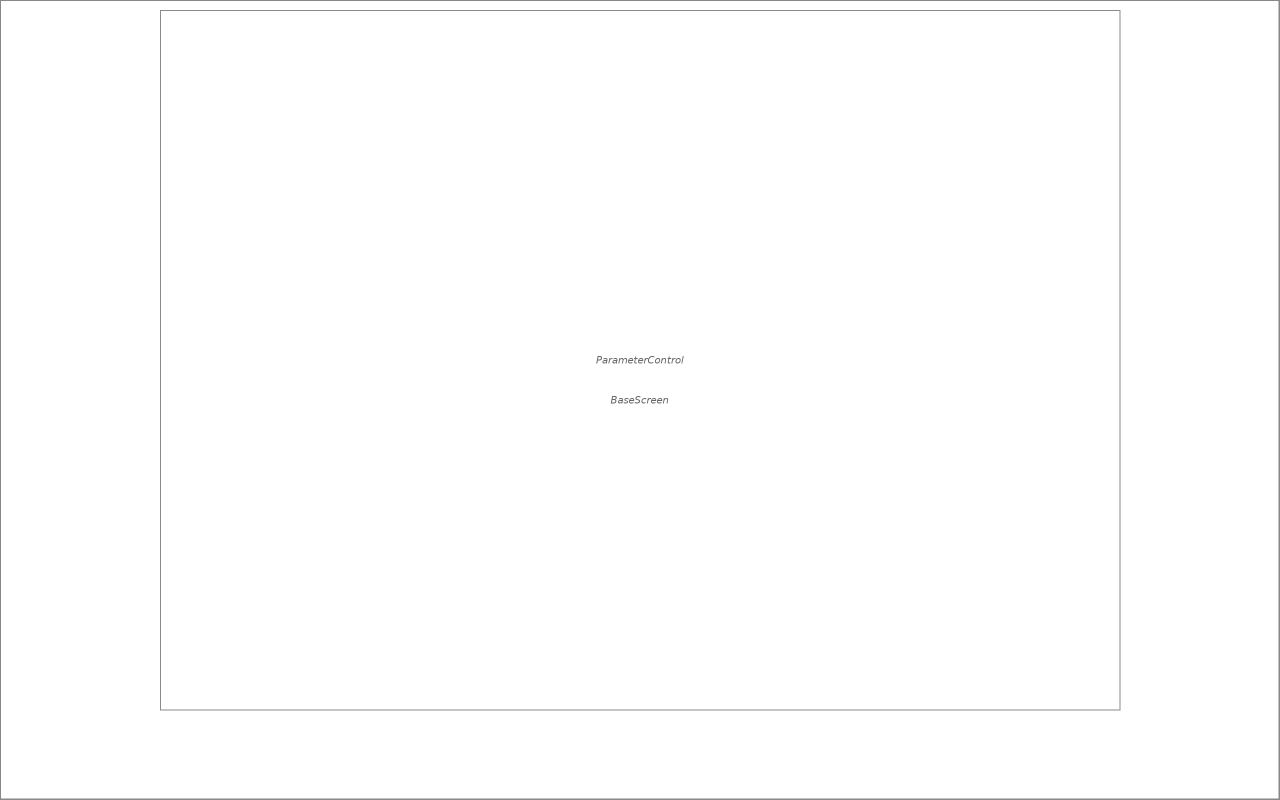
VISUALIZATION VISU_TEST  // 1280x800
    Frame (0,0 1280x800)
        shows BaseScreen(nFaultsInLog := GVL_Utilities.fbFaultHandler.nFaultsInLog)
    Frame (160,10 960x700)
        shows ParameterControl()
END_VISUALIZATION

(* stored: Version 1.1.0.1, ProductVersion 3.1.4024.11
   Visu VISU_TEST: Id {be5d7be9-6163-4e15-836c-0969efcf4b70} *)
